// TIA Portal V20 export
FUNCTION_BLOCK "Simulation"   // FB50062, LAD
// stored: MemoryReserve 100, Namespace Unit1.Em7, SetENOAutomatically false
   VAR_INPUT
      simulation { ExternalAccessible := 'False'; ExternalVisible := 'False'; ExternalWritable := 'False'} : Bool;
   END_VAR
   VAR
      instActuator { ExternalAccessible := 'False'; ExternalVisible := 'False'; ExternalWritable := 'False'} : Array[0..19] of "LER_SimActuator";
   END_VAR
   VAR_TEMP   // added for the SCL form of the ladder/FBD networks
      _w1 : Bool;
      _w2 : Bool;
      _w3 : Bool;
      _w4 : Bool;
      _w5 : Bool;
      _w6 : Bool;
   END_VAR
BEGIN

REGION Network 1: Two Way Actuator
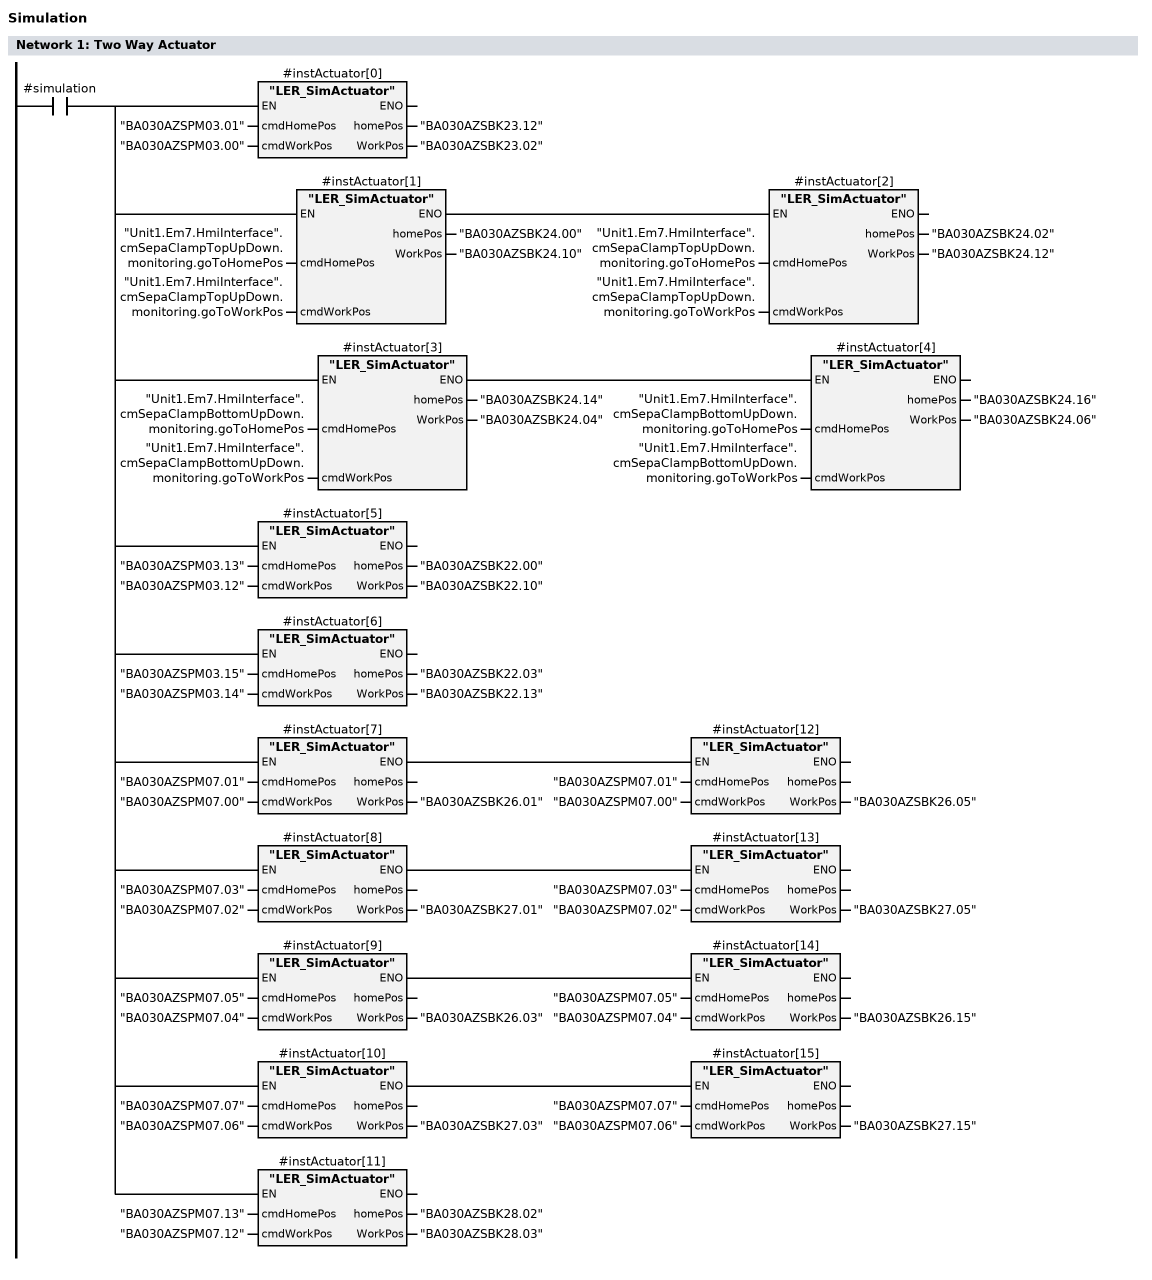
   RUNG wire#powerrail
      Contact( #simulation )
      wire#w1
      #instActuator[0](cmdHomePos := "BA030AZSPM03.01", cmdWorkPos := "BA030AZSPM03.00", homePos => "BA030AZSBK23.12", WorkPos => "BA030AZSBK23.02")
   END_RUNG
   RUNG wire#w1
      #instActuator[1](cmdHomePos := "Unit1.Em7.HmiInterface".cmSepaClampTopUpDown.monitoring.goToHomePos, cmdWorkPos := "Unit1.Em7.HmiInterface".cmSepaClampTopUpDown.monitoring.goToWorkPos, homePos => "BA030AZSBK24.00", WorkPos => "BA030AZSBK24.10")
      #instActuator[2](cmdHomePos := "Unit1.Em7.HmiInterface".cmSepaClampTopUpDown.monitoring.goToHomePos, cmdWorkPos := "Unit1.Em7.HmiInterface".cmSepaClampTopUpDown.monitoring.goToWorkPos, homePos => "BA030AZSBK24.02", WorkPos => "BA030AZSBK24.12")
   END_RUNG
   RUNG wire#w1
      #instActuator[3](cmdHomePos := "Unit1.Em7.HmiInterface".cmSepaClampBottomUpDown.monitoring.goToHomePos, cmdWorkPos := "Unit1.Em7.HmiInterface".cmSepaClampBottomUpDown.monitoring.goToWorkPos, homePos => "BA030AZSBK24.14", WorkPos => "BA030AZSBK24.04")
      #instActuator[4](cmdHomePos := "Unit1.Em7.HmiInterface".cmSepaClampBottomUpDown.monitoring.goToHomePos, cmdWorkPos := "Unit1.Em7.HmiInterface".cmSepaClampBottomUpDown.monitoring.goToWorkPos, homePos => "BA030AZSBK24.16", WorkPos => "BA030AZSBK24.06")
   END_RUNG
   RUNG wire#w1
      #instActuator[5](cmdHomePos := "BA030AZSPM03.13", cmdWorkPos := "BA030AZSPM03.12", homePos => "BA030AZSBK22.00", WorkPos => "BA030AZSBK22.10")
   END_RUNG
   RUNG wire#w1
      #instActuator[6](cmdHomePos := "BA030AZSPM03.15", cmdWorkPos := "BA030AZSPM03.14", homePos => "BA030AZSBK22.03", WorkPos => "BA030AZSBK22.13")
   END_RUNG
   RUNG wire#w1
      #instActuator[7](cmdHomePos := "BA030AZSPM07.01", cmdWorkPos := "BA030AZSPM07.00", homePos =>, WorkPos => "BA030AZSBK26.01")
      #instActuator[12](cmdHomePos := "BA030AZSPM07.01", cmdWorkPos := "BA030AZSPM07.00", homePos =>, WorkPos => "BA030AZSBK26.05")
   END_RUNG
   RUNG wire#w1
      #instActuator[8](cmdHomePos := "BA030AZSPM07.03", cmdWorkPos := "BA030AZSPM07.02", homePos =>, WorkPos => "BA030AZSBK27.01")
      #instActuator[13](cmdHomePos := "BA030AZSPM07.03", cmdWorkPos := "BA030AZSPM07.02", homePos =>, WorkPos => "BA030AZSBK27.05")
   END_RUNG
   RUNG wire#w1
      #instActuator[9](cmdHomePos := "BA030AZSPM07.05", cmdWorkPos := "BA030AZSPM07.04", homePos =>, WorkPos => "BA030AZSBK26.03")
      #instActuator[14](cmdHomePos := "BA030AZSPM07.05", cmdWorkPos := "BA030AZSPM07.04", homePos =>, WorkPos => "BA030AZSBK26.15")
   END_RUNG
   RUNG wire#w1
      #instActuator[10](cmdHomePos := "BA030AZSPM07.07", cmdWorkPos := "BA030AZSPM07.06", homePos =>, WorkPos => "BA030AZSBK27.03")
      #instActuator[15](cmdHomePos := "BA030AZSPM07.07", cmdWorkPos := "BA030AZSPM07.06", homePos =>, WorkPos => "BA030AZSBK27.15")
   END_RUNG
   RUNG wire#w1
      #instActuator[11](cmdHomePos := "BA030AZSPM07.13", cmdWorkPos := "BA030AZSPM07.12", homePos => "BA030AZSBK28.02", WorkPos => "BA030AZSBK28.03")
   END_RUNG
   // the same network as SCL:
   IF #simulation THEN
       #instActuator[0](cmdHomePos := "BA030AZSPM03.01",   // "LER_SimActuator"
                        cmdWorkPos := "BA030AZSPM03.00",
                        homePos => "BA030AZSBK23.12",
                        WorkPos => "BA030AZSBK23.02");
   END_IF;
   #instActuator[1](EN := #simulation,   // "LER_SimActuator"
                    cmdHomePos := "Unit1.Em7.HmiInterface".cmSepaClampTopUpDown.monitoring.goToHomePos,
                    cmdWorkPos := "Unit1.Em7.HmiInterface".cmSepaClampTopUpDown.monitoring.goToWorkPos,
                    homePos => "BA030AZSBK24.00",
                    WorkPos => "BA030AZSBK24.10",
                    ENO => #_w1);
   IF #_w1 THEN
       #instActuator[2](cmdHomePos := "Unit1.Em7.HmiInterface".cmSepaClampTopUpDown.monitoring.goToHomePos,   // "LER_SimActuator"
                        cmdWorkPos := "Unit1.Em7.HmiInterface".cmSepaClampTopUpDown.monitoring.goToWorkPos,
                        homePos => "BA030AZSBK24.02",
                        WorkPos => "BA030AZSBK24.12");
   END_IF;
   #instActuator[3](EN := #simulation,   // "LER_SimActuator"
                    cmdHomePos := "Unit1.Em7.HmiInterface".cmSepaClampBottomUpDown.monitoring.goToHomePos,
                    cmdWorkPos := "Unit1.Em7.HmiInterface".cmSepaClampBottomUpDown.monitoring.goToWorkPos,
                    homePos => "BA030AZSBK24.14",
                    WorkPos => "BA030AZSBK24.04",
                    ENO => #_w2);
   IF #_w2 THEN
       #instActuator[4](cmdHomePos := "Unit1.Em7.HmiInterface".cmSepaClampBottomUpDown.monitoring.goToHomePos,   // "LER_SimActuator"
                        cmdWorkPos := "Unit1.Em7.HmiInterface".cmSepaClampBottomUpDown.monitoring.goToWorkPos,
                        homePos => "BA030AZSBK24.16",
                        WorkPos => "BA030AZSBK24.06");
   END_IF;
   IF #simulation THEN
       #instActuator[5](cmdHomePos := "BA030AZSPM03.13",   // "LER_SimActuator"
                        cmdWorkPos := "BA030AZSPM03.12",
                        homePos => "BA030AZSBK22.00",
                        WorkPos => "BA030AZSBK22.10");
       #instActuator[6](cmdHomePos := "BA030AZSPM03.15",   // "LER_SimActuator"
                        cmdWorkPos := "BA030AZSPM03.14",
                        homePos => "BA030AZSBK22.03",
                        WorkPos => "BA030AZSBK22.13");
   END_IF;
   #instActuator[7](EN := #simulation,   // "LER_SimActuator"
                    cmdHomePos := "BA030AZSPM07.01",
                    cmdWorkPos := "BA030AZSPM07.00",
                    WorkPos => "BA030AZSBK26.01",
                    ENO => #_w3);
   IF #_w3 THEN
       #instActuator[12](cmdHomePos := "BA030AZSPM07.01",   // "LER_SimActuator"
                         cmdWorkPos := "BA030AZSPM07.00",
                         WorkPos => "BA030AZSBK26.05");
   END_IF;
   #instActuator[8](EN := #simulation,   // "LER_SimActuator"
                    cmdHomePos := "BA030AZSPM07.03",
                    cmdWorkPos := "BA030AZSPM07.02",
                    WorkPos => "BA030AZSBK27.01",
                    ENO => #_w4);
   IF #_w4 THEN
       #instActuator[13](cmdHomePos := "BA030AZSPM07.03",   // "LER_SimActuator"
                         cmdWorkPos := "BA030AZSPM07.02",
                         WorkPos => "BA030AZSBK27.05");
   END_IF;
   #instActuator[9](EN := #simulation,   // "LER_SimActuator"
                    cmdHomePos := "BA030AZSPM07.05",
                    cmdWorkPos := "BA030AZSPM07.04",
                    WorkPos => "BA030AZSBK26.03",
                    ENO => #_w5);
   IF #_w5 THEN
       #instActuator[14](cmdHomePos := "BA030AZSPM07.05",   // "LER_SimActuator"
                         cmdWorkPos := "BA030AZSPM07.04",
                         WorkPos => "BA030AZSBK26.15");
   END_IF;
   #instActuator[10](EN := #simulation,   // "LER_SimActuator"
                     cmdHomePos := "BA030AZSPM07.07",
                     cmdWorkPos := "BA030AZSPM07.06",
                     WorkPos => "BA030AZSBK27.03",
                     ENO => #_w6);
   IF #_w6 THEN
       #instActuator[15](cmdHomePos := "BA030AZSPM07.07",   // "LER_SimActuator"
                         cmdWorkPos := "BA030AZSPM07.06",
                         WorkPos => "BA030AZSBK27.15");
   END_IF;
   IF #simulation THEN
       #instActuator[11](cmdHomePos := "BA030AZSPM07.13",   // "LER_SimActuator"
                         cmdWorkPos := "BA030AZSPM07.12",
                         homePos => "BA030AZSBK28.02",
                         WorkPos => "BA030AZSBK28.03");
   END_IF;
END_REGION
END_FUNCTION_BLOCK
